PROGRAM P_Demo_LINT_TO_LARGE
VAR
    liNative : LINT := -123456789;
    liLegacy : T_LARGE_INTEGER;
    bConvert : BOOL;
END_VAR

// ============================================================
// Tc2_Utilities.LINT_TO_LARGE 演示程序（FUNCTION，单周期触发）
// ============================================================
// 场景：本地用 LINT 做算术，调用一个只接 T_LARGE_INTEGER 的旧 FB 前转一下。
// 价值：替代手写 SHR/AND/拼装。
// 验证步骤：
//   1. 把本 PROGRAM 加到 PlcTask 调用列表
//   2. 编译 + 登录
//   3. 在线把 b... 触发位置 TRUE 一个周期
//   4. 观察输出变量是否符合期望
// ============================================================

IF bConvert THEN
    liLegacy := LINT_TO_LARGE(liNative);
    bConvert := FALSE;
END_IF;

END_PROGRAM

(* stored: Version 1.1.0.1, ProductVersion 3.1.4024.5
   POU P_Demo_LINT_TO_LARGE: Id {1bbdb997-1c2a-5f12-9f19-735bcf704ca3}, SpecialFunc None *)
